TYPE E_PrintParamType :
(
	Undefined,
	Pressure,
	Feed,
	Flow,
	Frequency,
	Pulse,
	Voltage
)USINT;
END_TYPE

(* stored: Version 1.1.0.1, ProductVersion 3.1.4024.9
   DUT E_PrintParamType: Id {71e59337-501e-4b7d-b85e-1d0ab0154e8d} *)
